FUNCTION_BLOCK FB_TrafficLight
VAR_INPUT
	clear_road 			: BOOL;
	block_road 			: BOOL;
	disable_system		: BOOL;
END_VAR
VAR_OUTPUT
	red_light			: BOOL;
	yellow_light		: BOOL;
	green_light			: BOOL;
END_VAR
VAR
	// state variables
	currentState		: 	EN_TRAFFICLIGHT_STATE := EN_TRAFFICLIGHT_STATE.STATE_INIT;
	lastState			: 	EN_TRAFFICLIGHT_STATE := EN_TRAFFICLIGHT_STATE.STATE_UNDEFINED;
	timer				: 	TON;
	// flag to reset the timer after the state machine has used it
	resetTimer			:	BOOL;
	// flag to update last state
	transitionDone		: 	BOOL;
END_VAR

timer();  // call timer

// state machine
CASE currentState OF
	EN_TRAFFICLIGHT_STATE.STATE_UNDEFINED:
	// jump to init	
	currentState := EN_TRAFFICLIGHT_STATE.STATE_INIT;
	
	//*****************************//
	EN_TRAFFICLIGHT_STATE.STATE_INIT:
	// jump to red
	currentState := EN_TRAFFICLIGHT_STATE.STATE_RED;
	
	//*****************************//
	EN_TRAFFICLIGHT_STATE.STATE_RED:
	// entry action
	IF(currentState <> lastState) THEN
		// enable only red light
		red_light := TRUE; yellow_light := FALSE; green_light := FALSE;
		lastState := currentState;  // update last state
	END_IF
	
	// clear road (prio 2)
	IF(clear_road) THEN
		currentState := EN_TRAFFICLIGHT_STATE.STATE_RED_YELLOW;
	END_IF
	
	// clear road (prio 1)
	IF(disable_system) THEN
		currentState := EN_TRAFFICLIGHT_STATE.STATE_DISABLED;
	END_IF
	
	//*****************************//
	EN_TRAFFICLIGHT_STATE.STATE_RED_YELLOW:
	// entry action
	IF(currentState <> lastState) THEN
		// enable red and yellow light
		red_light := TRUE; yellow_light := TRUE; green_light := FALSE;
		lastState := currentState;  // update last state
	END_IF
	
	// start timer for automatic state change
	timer.PT := T#2S;
	timer.IN := TRUE;
	
	// timer finished => exit action
	IF timer.Q THEN
		currentState := EN_TRAFFICLIGHT_STATE.STATE_GREEN;
		resetTimer := TRUE;
	END_IF
	
	//*****************************//
	EN_TRAFFICLIGHT_STATE.STATE_YELLOW:
	// entry action
	IF(currentState <> lastState) THEN
		// enable yellow light only
		red_light := FALSE; yellow_light := TRUE; green_light := FALSE;
		lastState := currentState;  // update last state
	END_IF
	
	// start timer for automatic state change
	timer.PT := T#5S;
	timer.IN := TRUE;
	
	// timer finished => exit action
	IF timer.Q THEN
		currentState := EN_TRAFFICLIGHT_STATE.STATE_RED;
		resetTimer := TRUE;
	END_IF
	
	//*****************************//
	EN_TRAFFICLIGHT_STATE.STATE_GREEN:
	// entry action
	IF(currentState <> lastState) THEN
		// enable green light only
		red_light := FALSE; yellow_light := FALSE; green_light := TRUE;
		lastState := currentState;  // update last state
	END_IF
	
	// block_road signal
	IF(block_road) THEN
		currentState := EN_TRAFFICLIGHT_STATE.STATE_YELLOW;
	END_IF
	
	//*****************************//
	EN_TRAFFICLIGHT_STATE.STATE_DISABLED:
	// disable all lights
	red_light := FALSE; green_light := FALSE;
	
	// start timer for yellow blinking
	timer.PT := T#1S;
	timer.IN := TRUE;
	
	// invert yellow light (blink)
	IF timer.Q THEN
		yellow_light := NOT yellow_light;
		resetTimer := TRUE;
	END_IF
	
	// system was re-enabled 
	IF (disable_system = FALSE) THEN
		lastState := currentState;  // update last state
		currentState := EN_TRAFFICLIGHT_STATE.STATE_RED;
		resetTimer := TRUE;
	END_IF
	
END_CASE

// reset timer since it was used
IF resetTimer THEN
	timer.IN := FALSE;
	timer();  // call to trigger edge
	resetTimer := FALSE;	
END_IF

END_FUNCTION_BLOCK

(* stored: Version 1.1.0.1, ProductVersion 3.1.4024.9
   POU FB_TrafficLight: Id {5c204fba-31a4-4ff6-939b-a4b43b44ff6c}, SpecialFunc None *)
